FUNCTION_BLOCK PUBLIC FB_IndexedPosition

VAR
	// Configuration 		: ST_IndexedPositionConfiguration;
	Controls			: ST_IndexedPositionControls;
	// Status				: ST_IndexedPositionStatus;
	Links				: ST_IndexedPositionLinks;
END_VAR

_M_StateMachine();

// Broadcast Part Presence Status
Controls.Front.PartPresent := Controls.AreaMonitoring OR Controls.ArrivalDetection;
Controls.Rear.PartPresent := Controls.AreaMonitoring OR Controls.ArrivalDetection;
Controls.Left.PartPresent := Controls.AreaMonitoring OR Controls.ArrivalDetection;
Controls.Right.PartPresent := Controls.AreaMonitoring OR Controls.ArrivalDetection;

// Broadcast State
Controls.Front.State := Controls.State;
Controls.Rear.State := Controls.State;
Controls.Right.State := Controls.State;
Controls.Left.State := Controls.State;

// Propogate Directional Controls Request to recieve to main level
(*
IF Controls.Request =  E_IndexedPositionTransitionRequest.NoRequest (*AND Controls.State = E_IndexedPositionStates.Starved *)THEN
	IF Controls.Front.Request = E_IndexedPositionSimplifiedRequest.Recieve THEN
		Controls.Request :=  E_IndexedPositionTransitionRequest.ReceiveFromFront;
	ELSIF Controls.Rear.Request = E_IndexedPositionSimplifiedRequest.Recieve THEN
		Controls.Request :=  E_IndexedPositionTransitionRequest.ReceiveFromRear;
	ELSIF Controls.Right.Request = E_IndexedPositionSimplifiedRequest.Recieve THEN
		Controls.Request :=  E_IndexedPositionTransitionRequest.ReceiveFromRight;
	ELSIF Controls.Left.Request = E_IndexedPositionSimplifiedRequest.Recieve THEN
		Controls.Request :=  E_IndexedPositionTransitionRequest.ReceiveFromLeft;
	END_IF
END_IF
*)

// Links.Self.State := State;

METHOD PRIVATE _M_StateMachine : BOOL
VAR_INPUT
END_VAR
(*IF Configuration.BypassIndexedPosition THEN
	Controls.State := E_IndexedPositionStates.Bypass;
ELSE
	Controls.State := E_IndexedPositionStates.Idle;
END_IF*)

CASE Controls.State OF
	E_IndexedPositionStates.Starved:
		// Command 
		Controls.Request 	:= E_IndexedPositionTransitionRequest.NoRequest;
		// Error Handling
		
		// Branch Conditions
		IF NOT Controls.AreaMonitoring AND NOT Controls.ArrivalDetection THEN
			
		   	IF __ISVALIDREF(Links.Rear) THEN
				IF Links.Rear.Request = E_IndexedPositionSimplifiedRequest.Send THEN
					Controls.State 			:= E_IndexedPositionStates.ReceivingFromRear;
					Controls.Rear.Request 	:= E_IndexedPositionSimplifiedRequest.Recieve;
					// Controls.Request	 	:= E_IndexedPositionTransitionRequest.ReceiveFromRear;
				END_IF
				
			ELSIF __ISVALIDREF(Links.Front) THEN
				IF  Links.Front.Request = E_IndexedPositionSimplifiedRequest.Send THEN
					Controls.State 			:= E_IndexedPositionStates.ReceivingFromFront;
					Controls.Front.Request 	:= E_IndexedPositionSimplifiedRequest.Recieve;
					// Controls.Request	 	:= E_IndexedPositionTransitionRequest.ReceiveFromFront;
				END_IF
			
			ELSIF __ISVALIDREF(Links.Left) THEN
				IF  Links.Left.Request = E_IndexedPositionSimplifiedRequest.Send THEN
					Controls.State 			:= E_IndexedPositionStates.ReceivingFromLeft;
					Controls.Left.Request 	:= E_IndexedPositionSimplifiedRequest.Recieve;
					// Controls.Request	 	:= E_IndexedPositionTransitionRequest.ReceiveFromLeft;
				END_IF
			
			ELSIF __ISVALIDREF(Links.Right) THEN
				IF   Links.Right.Request = E_IndexedPositionSimplifiedRequest.Send THEN
					Controls.State 			:= E_IndexedPositionStates.ReceivingFromRight;
					Controls.Right.Request 	:= E_IndexedPositionSimplifiedRequest.Recieve;
					// Controls.Request	 	:= E_IndexedPositionTransitionRequest.ReceiveFromRight;
				END_IF
				
			END_IF
			
		ELSIF Controls.AreaMonitoring AND Controls.Request = E_IndexedPositionTransitionRequest.NoRequest THEN
			Controls.State 			:= E_IndexedPositionStates.Idle;
			// Controls.Request	 	:= E_IndexedPositionTransitionRequest.NoRequest;
		END_IF
		
	E_IndexedPositionStates.Idle:
			
		// Error Handling
		
		// Branch Conditions
		IF Controls.AreaMonitoring AND Controls.ArrivalDetection THEN
			// Link Request for Handshake
			IF Controls.Request = E_IndexedPositionTransitionRequest.SendToFront THEN
				Controls.Front.Request := E_IndexedPositionSimplifiedRequest.Send;
			ELSIF Controls.Request = E_IndexedPositionTransitionRequest.SendToLeft THEN
				Controls.Left.Request 	:= E_IndexedPositionSimplifiedRequest.Send;
			ELSIF Controls.Request = E_IndexedPositionTransitionRequest.SendToRear THEN
				Controls.Rear.Request 	:= E_IndexedPositionSimplifiedRequest.Send;
			ELSIF Controls.Request = E_IndexedPositionTransitionRequest.SendToRight THEN
				Controls.Right.Request := E_IndexedPositionSimplifiedRequest.Send;
			END_IF
		
			IF Controls.Request = E_IndexedPositionTransitionRequest.SendToFront THEN
				IF __ISVALIDREF(Links.Front) THEN
					IF NOT Links.Front.PartPresent AND
					   Links.Front.Request = E_IndexedPositionSimplifiedRequest.Recieve THEN
						  
						Controls.State 			:= E_IndexedPositionStates.SendingToFront;
						Controls.Front.Request 	:= E_IndexedPositionSimplifiedRequest.NoRequest;
						Links.Front.Request 	:= E_IndexedPositionSimplifiedRequest.NoRequest;
						
					ELSIF Links.Front.PartPresent OR 
						  Links.Front.Request <> E_IndexedPositionSimplifiedRequest.Recieve OR
						  Links.Front.State <> E_IndexedPositionStates.Starved THEN
						  
						Controls.State := E_IndexedPositionStates.Blocked;
						
					END_IF
				END_IF
			
			ELSIF Controls.Request = E_IndexedPositionTransitionRequest.SendToLeft THEN
				IF __ISVALIDREF(Links.Left) THEN
					IF NOT Links.Left.PartPresent AND 
						  Links.Left.Request = E_IndexedPositionSimplifiedRequest.Recieve THEN
						  
						Controls.State 			:= E_IndexedPositionStates.SendingToLeft;
						Controls.Left.Request 	:= E_IndexedPositionSimplifiedRequest.NoRequest;
						Links.Left.Request 		:= E_IndexedPositionSimplifiedRequest.NoRequest;
						
					ELSIF Links.Left.PartPresent OR 
						  Links.Left.Request <> E_IndexedPositionSimplifiedRequest.Recieve OR
						  Links.Left.State <> E_IndexedPositionStates.Starved THEN
						  
						Controls.State := E_IndexedPositionStates.Blocked;
						
					END_IF
				END_IF
				
			ELSIF Controls.Request = E_IndexedPositionTransitionRequest.SendToRear THEN
				IF __ISVALIDREF(Links.Rear) THEN
					IF NOT Links.Rear.PartPresent AND
					   Links.Rear.Request = E_IndexedPositionSimplifiedRequest.Recieve THEN
						  
						Controls.State 			:= E_IndexedPositionStates.SendingToRear;
						Controls.Rear.Request 	:= E_IndexedPositionSimplifiedRequest.NoRequest;
						Links.Rear.Request 		:= E_IndexedPositionSimplifiedRequest.NoRequest;
						
					ELSIF Links.Rear.PartPresent OR 
						  Links.Rear.Request <> E_IndexedPositionSimplifiedRequest.Recieve OR 
						  Links.Rear.State <> E_IndexedPositionStates.Starved THEN
						  
						Controls.State := E_IndexedPositionStates.Blocked;
						
					END_IF
				END_IF
				
			ELSIF Controls.Request = E_IndexedPositionTransitionRequest.SendToRight THEN
				IF __ISVALIDREF(Links.Right) THEN
					IF NOT Links.Right.PartPresent AND
					   Links.Right.Request = E_IndexedPositionSimplifiedRequest.Recieve THEN
						  
						Controls.State 			:= E_IndexedPositionStates.SendingToRight;
						Controls.Right.Request 	:= E_IndexedPositionSimplifiedRequest.NoRequest;
						Links.Right.Request 	:= E_IndexedPositionSimplifiedRequest.NoRequest;
						
					ELSIF Links.Right.PartPresent OR 
						  Links.Right.Request <> E_IndexedPositionSimplifiedRequest.Recieve OR
						  Links.Right.State <> E_IndexedPositionStates.Starved THEN
						  
						Controls.State := E_IndexedPositionStates.Blocked;
						
					END_IF
				END_IF
				
			END_IF
			
		ELSIF NOT Controls.AreaMonitoring AND NOT Controls.ArrivalDetection AND Controls.Request = E_IndexedPositionTransitionRequest.NoRequest THEN
			Controls.State 		:= E_IndexedPositionStates.Starved;
			Controls.Request 	:= E_IndexedPositionTransitionRequest.NoRequest;
			
		ELSIF Controls.AreaMonitoring OR Controls.ArrivalDetection  THEN
			//
		END_IF
	
	E_IndexedPositionStates.Blocked:
		// Command
		// Controls.Request 	:= E_IndexedPositionTransitionRequest.NoRequest;
		// Error Handling
		
		// Branch Conditions
		IF Controls.AreaMonitoring AND Controls.ArrivalDetection  THEN
			IF __ISVALIDREF(Links.Front) THEN
				IF Controls.Request = E_IndexedPositionTransitionRequest.SendToFront AND 
				   NOT Links.Front.PartPresent AND 
				   Links.Front.Request = E_IndexedPositionSimplifiedRequest.Recieve THEN
						
				   	Controls.State := E_IndexedPositionStates.Idle;
				END_IF
				
			ELSIF __ISVALIDREF(Links.Left) THEN
				IF Controls.Request = E_IndexedPositionTransitionRequest.SendToLeft AND 
			       NOT Links.Left.PartPresent AND 
				   Links.Left.Request = E_IndexedPositionSimplifiedRequest.Recieve THEN
				  
					Controls.State := E_IndexedPositionStates.Idle;
				END_IF
				
			ELSIF __ISVALIDREF(Links.Rear) THEN
				IF Controls.Request = E_IndexedPositionTransitionRequest.SendToRear AND 
			       NOT Links.Rear.PartPresent AND 
				   Links.Rear.Request = E_IndexedPositionSimplifiedRequest.Recieve THEN
				  
					Controls.State := E_IndexedPositionStates.Idle;
				END_IF
				
			ELSIF __ISVALIDREF(Links.Right) THEN
				IF Controls.Request = E_IndexedPositionTransitionRequest.SendToRight AND 
			       NOT Links.Right.PartPresent AND 
				   Links.Right.Request = E_IndexedPositionSimplifiedRequest.Recieve THEN
				  
					Controls.State := E_IndexedPositionStates.Idle;
				END_IF
				
			END_IF
			
		ELSIF NOT Controls.AreaMonitoring AND NOT Controls.ArrivalDetection  THEN
			// Starved or Error?
		END_IF
	
	E_IndexedPositionStates.ReceivingFromLeft,
	E_IndexedPositionStates.ReceivingFromRight,
	E_IndexedPositionStates.ReceivingFromFront,
	E_IndexedPositionStates.ReceivingFromRear:
		// Command
		
		// Error Handling
		
		// Branch Conditions
		IF Controls.ArrivalDetection THEN
			Controls.State 		:= E_IndexedPositionStates.Idle;
		END_IF
	
	E_IndexedPositionStates.SendingToLeft:
		// Command
		
		// Error Handling
		
		// Branch Conditions
		IF __ISVALIDREF(Links.Left) THEN
			IF Links.Left.State = E_IndexedPositionStates.Idle THEN
				Controls.State 		:= E_IndexedPositionStates.Starved;
			END_IF
		END_IF
	
	E_IndexedPositionStates.SendingToRight:
		// Command
		
		// Error Handling
		
		// Branch Conditions
		IF __ISVALIDREF(Links.Right) THEN
			IF Links.Right.State = E_IndexedPositionStates.Idle THEN
				Controls.State 		:= E_IndexedPositionStates.Starved;
			END_IF
		END_IF
		
	E_IndexedPositionStates.SendingToFront:
		// Command
		
		// Error Handling
		
		// Branch Conditions
		IF __ISVALIDREF(Links.Front) THEN
			IF Links.Front.State = E_IndexedPositionStates.Idle THEN
				Controls.State 		:= E_IndexedPositionStates.Starved;
			END_IF
		END_IF
		
	E_IndexedPositionStates.SendingToRear:
		// Command
		
		// Error Handling
		
		// Branch Conditions
		IF __ISVALIDREF(Links.Rear) THEN
			IF Links.REar.State = E_IndexedPositionStates.Idle THEN
				Controls.State 		:= E_IndexedPositionStates.Starved;
			END_IF
		END_IF
		
	E_IndexedPositionStates.Bypass:
		Controls.Request := E_IndexedPositionTransitionRequest.NoRequest;
		
	E_IndexedPositionStates.Fault:
		// Command
		Controls.Request := E_IndexedPositionTransitionRequest.NoRequest;
		
		// Error Handling
		
		// Branch Conditions
	
END_CASE
END_METHOD

PROPERTY PUBLIC P_Controls : REFERENCE TO ST_IndexedPositionControls
GET
P_Controls REF= Controls;
END_GET
END_PROPERTY

PROPERTY PUBLIC P_Links : REFERENCE TO ST_IndexedPositionLinks
GET
P_Links REF= Links;
END_GET
END_PROPERTY

END_FUNCTION_BLOCK

(* stored: Version 1.1.0.1, ProductVersion 3.1.4024.12
   POU FB_IndexedPosition: Id {2f1b5667-a0f3-4b1e-97a1-207ac542be5f}, SpecialFunc None
   Method _M_StateMachine: Id {da0ce787-3a30-4396-967f-e071a2d629b3}
   Property P_Controls: Id {b310475e-32bc-40cf-a46b-4cc5dc485c1e}
   Get Get: Id {c32935fb-0864-43ce-9559-b349cd738359}
   Property P_Links: Id {9c6e14f0-9efa-4a56-b650-b0b8105c5a3a}
   Get Get: Id {908fadfb-bdbe-4eb2-90c4-0ea32058fac0} *)
